# EPICS autosave request: utcaApp/Db/ebpm_single.req
file "fmc_active_clk.req", P=${P}, R=${R}
file "fmc_adc_common.req", P=${P}, R=${R}
